{attribute 'GeneratedUsingTerminal: EPP6002-0002-0016'}
{attribute addProperty BoxType "EPP6002-0002-0016"}
{attribute addProperty Id "COM_TxPDO_Map_Inputs_Channel_1AT %I*COM_TxPDO_Map_Inputs_Channel_C252EAC224COM_TxPDO_Map_Inputs_Channel_2AT %I*COM_TxPDO_Map_Inputs_Channel_C252EAC224COM_RxPDO_Map_Outputs_Channel_1AT %Q*COM_RxPDO_Map_Outputs_Channel_B336F4EE24COM_RxPDO_Map_Outputs_Channel_2AT %Q*COM_RxPDO_Map_Outputs_Channel_B336F4EE24WcStateAT %I*WcState_9091E0EB2InfoDataAT %I*InfoData_94A18F5E2"}
{attribute addProperty CRC "3883112130"}
{attribute addProperty Size "100"}
TYPE EPP6002_E77396C2 EXTENDS EtcSlaveTerminalBase_947E5A46 :
STRUCT
	{attribute addProperty Name "COM_TxPDO_Map_Inputs_Channel_1"}
	COM_TxPDO_Map_Inputs_Channel_1 : COM_TxPDO_Map_Inputs_Channel_C252EAC2;
	{attribute addProperty Name "COM_TxPDO_Map_Inputs_Channel_2"}
	COM_TxPDO_Map_Inputs_Channel_2 : COM_TxPDO_Map_Inputs_Channel_C252EAC2;
	{attribute addProperty Name "COM_RxPDO_Map_Outputs_Channel_1"}
	COM_RxPDO_Map_Outputs_Channel_1 : COM_RxPDO_Map_Outputs_Channel_B336F4EE;
	{attribute addProperty Name "COM_RxPDO_Map_Outputs_Channel_2"}
	COM_RxPDO_Map_Outputs_Channel_2 : COM_RxPDO_Map_Outputs_Channel_B336F4EE;
	{attribute addProperty Name "WcState"}
	WcState : WcState_9091E0EB;
	{attribute addProperty Name "InfoData"}
	InfoData : InfoData_94A18F5E;
END_STRUCT
END_TYPE

(* stored: Version 1.2.0.0, ProductVersion 3.1.4024.9
   DUT EPP6002_E77396C2: Id {19c2b586-12b7-4d9c-8e5e-5ff5d73219b6} *)
